{attribute 'GeneratedUsingTerminal: CPXXXX-BK7902-0016'}
{attribute addProperty BoxType "CPXXXX-BK7902-0016"}
{attribute addProperty Id "Term_382_KL1002KL1002_BB38DA8F0"}
{attribute addProperty CRC "3434957117"}
{attribute addProperty Size "0"}
TYPE A_0009_CPXXXX_BK1150_0016_CCBD493D EXTENDS CPXXXX_13409EDF :
STRUCT
	{attribute addProperty Name "Term_382_KL1002"}
	Term_382_KL1002 : KL1002_BB38DA8F;
END_STRUCT
END_TYPE

(* stored: Version 1.2.0.0, ProductVersion 3.1.4024.9
   DUT A_0009_CPXXXX_BK1150_0016_CCBD493D: Id {e7d6bd31-355a-4a67-9f1c-96c4a721fc12} *)
